FUNCTION_BLOCK _TcoComponent EXTENDS TcoCore.TcoComponent
VAR
    _task : TcoTaskTest(THIS^);
    _serviceModeCount : ULINT;
END_VAR

_task();

{attribute 'TcRpcEnable'}
METHOD INTERNAL CallBodyFromTest
_task();
END_METHOD

(*~
    <docu>
        <summary>
            Restores this instance to the Ready state. Can be called explicitly or from within one of the restore mechanisms.
        </summary>
    </docu>
~*)
METHOD Restore : ITcoRestorable
_task.Restore();
END_METHOD

METHOD PROTECTED ServiceMode
_serviceModeCount := _serviceModeCount + 1;
END_METHOD

END_FUNCTION_BLOCK

(* stored: Version 1.1.0.1
   POU _TcoComponent: Id {b8956c28-5b21-0376-1161-3d340b13164a}, SpecialFunc None
   Method CallBodyFromTest: Id {e92a11df-7552-0d51-238d-48276d2fa228}
   Method Restore: Id {e7dc75ab-2cd2-0951-2512-113a4f119ffc}
   Method ServiceMode: Id {3fb21668-8b85-0a76-3335-10fe97bcba0c} *)
